FUNCTION TryConvert_UINT_TO_SINT : BOOL
VAR_INPUT
	in : UINT;
	out : REFERENCE TO SINT;
END_VAR

IF in > DatatypeLimits.MAX_VALUE_OF_UINT_WHICH_CAN_BE_HELD_IN_A_SINT THEN
	RETURN;
END_IF

out := UINT_TO_SINT(in);
TryConvert_UINT_TO_SINT := TRUE;

END_FUNCTION

(* stored: Version 1.1.0.1, ProductVersion 3.1.4024.12
   POU TryConvert_UINT_TO_SINT: Id {00bc5b1f-53e3-42f6-a7cf-c5229876fa5e}, SpecialFunc None *)
